SUBAPPLICATION AUI_AUI_MUX_2_VAL (* 2-Wege-Multiplexer fuer AUI/UINT-Werte mit 2 internen initval_AUI und AUI_MUX_2 / AUI_AUI_MUX_2. Schaltet per Event-Input (EI1, EI2) zwischen val1, val2 um. *)
  (* Standard: 61499-2; Description: Copyright (c) 2026 Meisterschulen am Ostbahnhof This program and the accompanying materials are made available under the terms of the Eclipse Public License 2.0 which is available at https://www.eclipse.org/legal/epl-2.0/ SPDX-License-Identifier: EPL-2.0 *)
  (* Version 1.0, 2026-09-10, Franz Höpfinger, Meisterschulen am Ostbahnhof, 2-fach AUI/UINT MUX mit initval *)
  PACKAGE MyLib::sys;
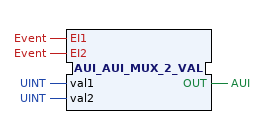
  EVENT_INPUT
    EI1; (* Event zur Auswahl von val1 *)
    EI2; (* Event zur Auswahl von val2 *)
  END_EVENT
  VAR_INPUT
    val1 : UINT; (* Initialer Ausgabewert bei EI1 *)
    val2 : UINT; (* Initialer Ausgabewert bei EI2 *)
  END_VAR
  PLUGS
    OUT : adapter::types::unidirectional::AUI; (* Ausgewaehlter AUI-Adapter Output *)
  END_PLUGS
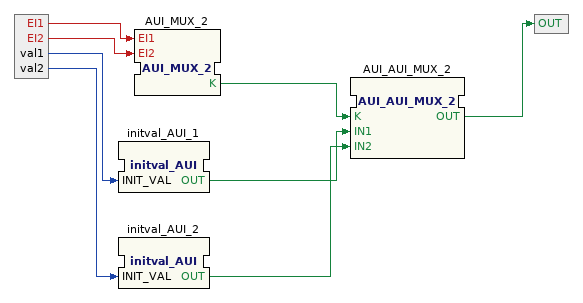
  FBS
    AUI_MUX_2 : adapter::events::unidirectional::AUI_MUX_2;
    AUI_AUI_MUX_2 : adapter::selection::unidirectional::AUI_AUI_MUX_2;
    initval_AUI_1 : adapter::types::unidirectional::AUI::initval::initval_AUI;
    initval_AUI_2 : adapter::types::unidirectional::AUI::initval::initval_AUI;
  END_FBS
  EVENT_CONNECTIONS
    EI1 TO AUI_MUX_2.EI1;
    EI2 TO AUI_MUX_2.EI2;
  END_CONNECTIONS
  DATA_CONNECTIONS
    val1 TO initval_AUI_1.INIT_VAL;
    val2 TO initval_AUI_2.INIT_VAL;
  END_CONNECTIONS
  ADAPTER_CONNECTIONS
    AUI_MUX_2.K TO AUI_AUI_MUX_2.K;
    initval_AUI_1.OUT TO AUI_AUI_MUX_2.IN1;
    initval_AUI_2.OUT TO AUI_AUI_MUX_2.IN2;
    AUI_AUI_MUX_2.OUT TO OUT;
  END_CONNECTIONS
END_SUBAPPLICATION
